(* Logix 5000 project; controller GEA_Test_Chamber vendor 1 type 14 code 196 rev 32.14; software revision 32.04; part 4 of 11 *)
(* tags used below, declared in another part *)
   Transaction : raC_UDT_ModbusClientTransaction;
   Wrk_Bit : DINT;
   Wrk_Byte : DINT;
(* raC_Tec_NetModbusTCPClient_BuildReqStr, continued *)

ROUTINE Prescan   (* ladder *)
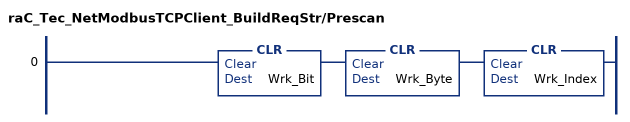
   0: CLR(Wrk_Bit)CLR(Wrk_Byte)CLR(Wrk_Index);
END_ROUTINE
END_ADD_ON_INSTRUCTION

ADD_ON_INSTRUCTION raC_Tec_NetModbusTCPClient_ChkWrReply   (* revision 2.0, ExecutePrescan *)
VAR_OUTPUT
   TransFound : BOOL; {access Read Only}
END_VAR
VAR_IN_OUT
   Transactions : raC_UDT_ModbusClientTransaction[5]; {required}
END_VAR
VAR_INPUT
   TransactionID : INT; {required}
   ModbusBytes : DINT; {required}
END_VAR
VAR_OUTPUT
   LocalOffset : INT; {access Read Only}
   Count : INT; {access Read Only}
END_VAR
VAR_INPUT
   Command : DINT; {required}
   LastTransaction : DINT; {required}
END_VAR
VAR
   Wrk_TransactionPtr : DINT; {access None}
END_VAR

ROUTINE Logic   (* ladder *)
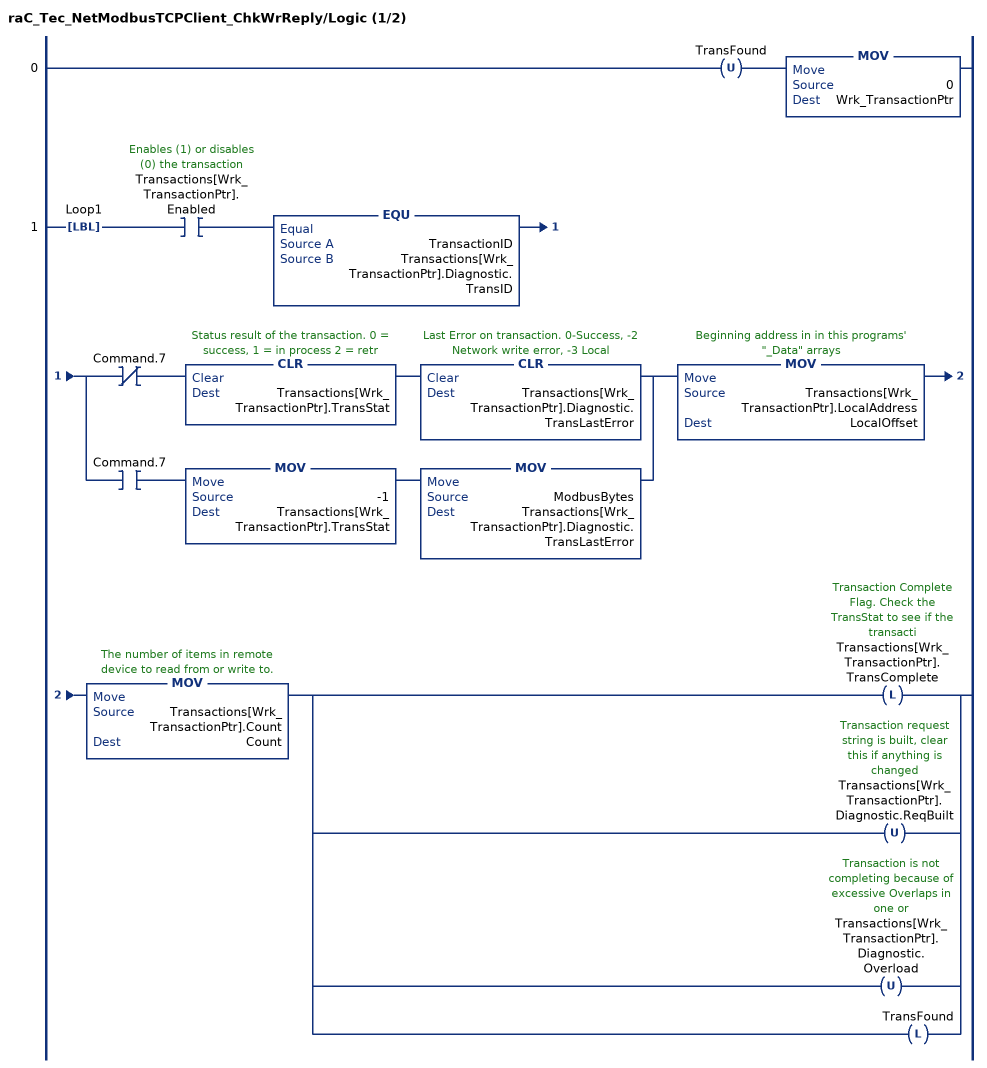
   0: OTU(TransFound)MOV(0,Wrk_TransactionPtr);
   1: LBL(Loop1)XIC(Transactions[Wrk_TransactionPtr].Enabled)EQU(TransactionID,Transactions[Wrk_TransactionPtr].Diagnostic.TransID)[XIO(Command.7) CLR(Transactions[Wrk_TransactionPtr].TransStat) CLR(Transactions[Wrk_TransactionPtr].Diagnostic.TransLastError) ,XIC(Command.7) MOV(-1,Transactions[Wrk_TransactionPtr].TransStat) MOV(ModbusBytes,Transactions[Wrk_TransactionPtr].Diagnostic.TransLastError) ]MOV(Transactions[Wrk_TransactionPtr].LocalAddress,LocalOffset)MOV(Transactions[Wrk_TransactionPtr].Count,Count)[OTL(Transactions[Wrk_TransactionPtr].TransComplete) ,OTU(Transactions[Wrk_TransactionPtr].Diagnostic.ReqBuilt) ,OTU(Transactions[Wrk_TransactionPtr].Diagnostic.Overload) ,OTL(TransFound) ];
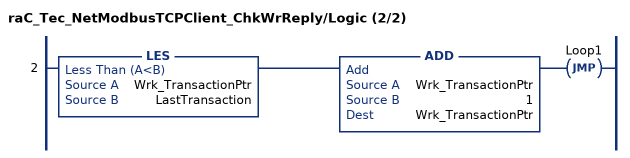
   2: LES(Wrk_TransactionPtr,LastTransaction)ADD(Wrk_TransactionPtr,1,Wrk_TransactionPtr)JMP(Loop1);
END_ROUTINE

ROUTINE Prescan   (* ladder *)
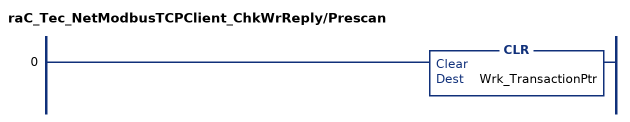
   0: CLR(Wrk_TransactionPtr);
END_ROUTINE
END_ADD_ON_INSTRUCTION

ADD_ON_INSTRUCTION raC_Tec_NetModbusTCPClient_RespStrBit   (* revision 2.0, ExecutePrescan *)
VAR_INPUT
   Inputs : BOOL; {required}
   Modbus_CMD_Len : INT; {required}
   LocalOffset : INT; {required}
END_VAR
VAR_IN_OUT
   ModbusData : raC_UDT_ModbusClientData; {required}
   CommandString : STR0462; {required}
END_VAR
VAR
   Wrk_BufferByteIndex : DINT; {access None}
   Wrk_Cmd_Last : INT; {access None}
   Wrk_Index : DINT; {access None}
   Wrk_BufferBitIndex : DINT; {access None}
   Wrk_ArraySize : DINT; {access None}
END_VAR

ROUTINE Logic   (* ladder *)
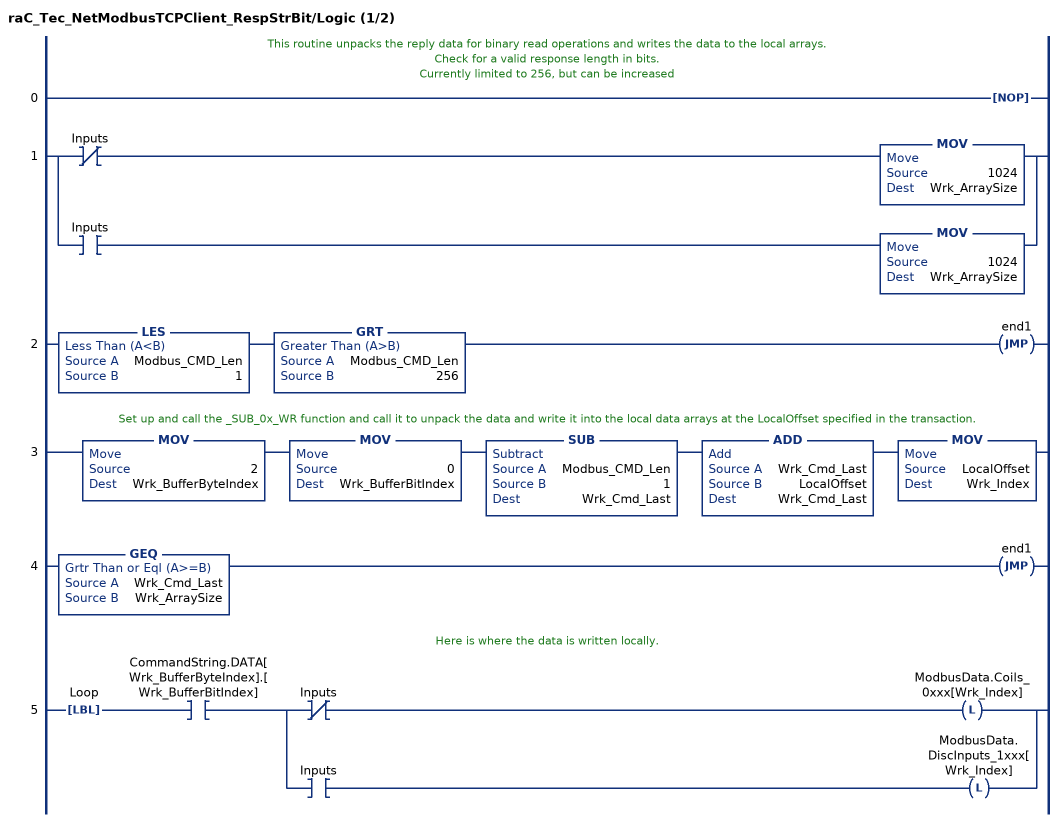
   // This routine unpacks the reply data for binary read operations and writes the data to the local arrays.
   // Check for a valid response length in bits.
   // Currently limited to 256, but can be increased
   0: NOP();
   1: [XIO(Inputs) MOV(1024,Wrk_ArraySize) ,XIC(Inputs) MOV(1024,Wrk_ArraySize) ];
   2: LES(Modbus_CMD_Len,1)GRT(Modbus_CMD_Len,256)JMP(end1);
   // Set up and call the _SUB_0x_WR function and call it to unpack the data and write it into the local data arrays at the LocalOffset specified in the transaction.
   3: MOV(2,Wrk_BufferByteIndex)MOV(0,Wrk_BufferBitIndex)SUB(Modbus_CMD_Len,1,Wrk_Cmd_Last)ADD(Wrk_Cmd_Last,LocalOffset,Wrk_Cmd_Last)MOV(LocalOffset,Wrk_Index);
   4: GEQ(Wrk_Cmd_Last,Wrk_ArraySize)JMP(end1);
   // Here is where the data is written locally.
   5: LBL(Loop)XIC(CommandString.DATA[Wrk_BufferByteIndex].[Wrk_BufferBitIndex])[XIO(Inputs) OTL(ModbusData.Coils_0xxx[Wrk_Index]) ,XIC(Inputs) OTL(ModbusData.DiscInputs_1xxx[Wrk_Index]) ];
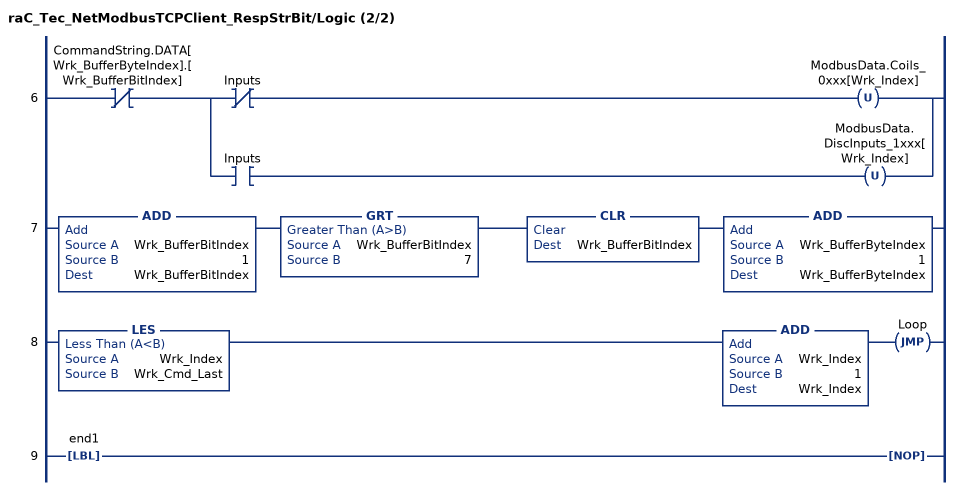
   6: XIO(CommandString.DATA[Wrk_BufferByteIndex].[Wrk_BufferBitIndex])[XIO(Inputs) OTU(ModbusData.Coils_0xxx[Wrk_Index]) ,XIC(Inputs) OTU(ModbusData.DiscInputs_1xxx[Wrk_Index]) ];
   7: ADD(Wrk_BufferBitIndex,1,Wrk_BufferBitIndex)GRT(Wrk_BufferBitIndex,7)CLR(Wrk_BufferBitIndex)ADD(Wrk_BufferByteIndex,1,Wrk_BufferByteIndex);
   8: LES(Wrk_Index,Wrk_Cmd_Last)ADD(Wrk_Index,1,Wrk_Index)JMP(Loop);
   9: LBL(end1)NOP();
END_ROUTINE

ROUTINE Prescan   (* ladder *)
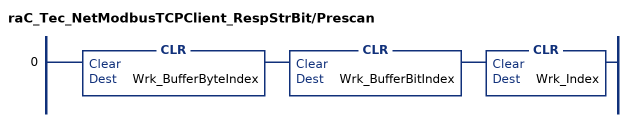
   0: CLR(Wrk_BufferByteIndex)CLR(Wrk_BufferBitIndex)CLR(Wrk_Index);
END_ROUTINE
END_ADD_ON_INSTRUCTION

ADD_ON_INSTRUCTION raC_Tec_NetModbusTCPClient_RespStrWord   (* revision 2.0, ExecutePrescan *)
VAR_INPUT
   Reg3xx : BOOL; {required}
   Modbus_CMD_Len : INT; {required}
   LocalOffset : INT; {required}
END_VAR
VAR_IN_OUT
   ModbusData : raC_UDT_ModbusClientData; {required}
   CommandString : STR0462; {required}
END_VAR
VAR
   Wrk_StringPosition : DINT; {access None}
   Wrk_Cmd_Last : INT; {access None}
   Wrk_Temp_Int : INT; {access None}
   Wrk_Index : DINT; {access None}
END_VAR

ROUTINE Logic   (* ladder *)
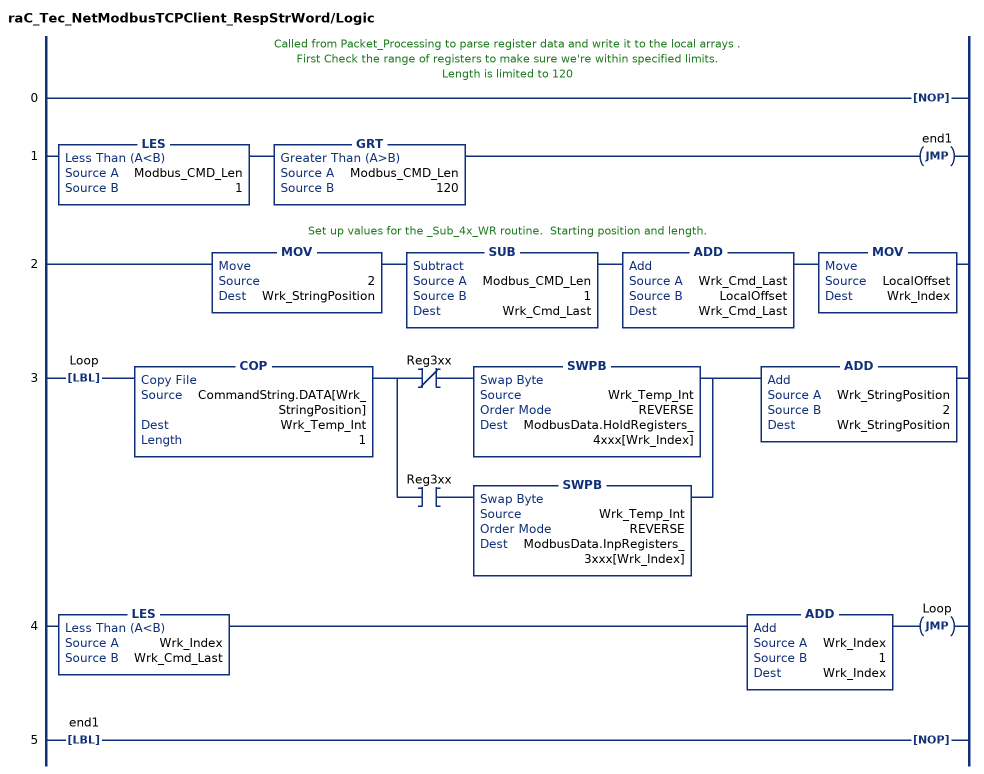
   // Called from Packet_Processing to parse register data and write it to the local arrays .
   // First Check the range of registers to make sure we're within specified limits.
   // Length is limited to 120
   0: NOP();
   1: LES(Modbus_CMD_Len,1)GRT(Modbus_CMD_Len,120)JMP(end1);
   // Set up values for the _Sub_4x_WR routine.  Starting position and length.
   2: MOV(2,Wrk_StringPosition)SUB(Modbus_CMD_Len,1,Wrk_Cmd_Last)ADD(Wrk_Cmd_Last,LocalOffset,Wrk_Cmd_Last)MOV(LocalOffset,Wrk_Index);
   3: LBL(Loop)COP(CommandString.DATA[Wrk_StringPosition],Wrk_Temp_Int,1)[XIO(Reg3xx) SWPB(Wrk_Temp_Int,REVERSE,ModbusData.HoldRegisters_4xxx[Wrk_Index]) ,XIC(Reg3xx) SWPB(Wrk_Temp_Int,REVERSE,ModbusData.InpRegisters_3xxx[Wrk_Index]) ]ADD(Wrk_StringPosition,2,Wrk_StringPosition);
   4: LES(Wrk_Index,Wrk_Cmd_Last)ADD(Wrk_Index,1,Wrk_Index)JMP(Loop);
   5: LBL(end1)NOP();
END_ROUTINE

ROUTINE Prescan   (* ladder *)
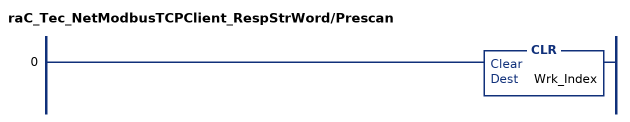
   0: CLR(Wrk_Index);
END_ROUTINE
END_ADD_ON_INSTRUCTION

ADD_ON_INSTRUCTION raC_Tec_NetModbusTCPServer_FndEmptySckt   (* revision 2.3 *)
VAR_INPUT
   NewInstance : DINT; {required}
   NewAddress : DINT; {required}
END_VAR
VAR_IN_OUT
   Sockets : raC_UDT_ModbusServerRWSocket[10]; {required}
END_VAR
VAR_OUTPUT
   Assigned : BOOL; {access Read Only, visible}
   NoRoom : BOOL; {access Read Only, visible}
END_VAR
VAR
   Wrk_InstIndex : DINT; {access None}
   Wrk_Size : DINT; {access None}
   Wrk_LastElement : DINT; {access None}
END_VAR

ROUTINE Logic   (* ladder *)
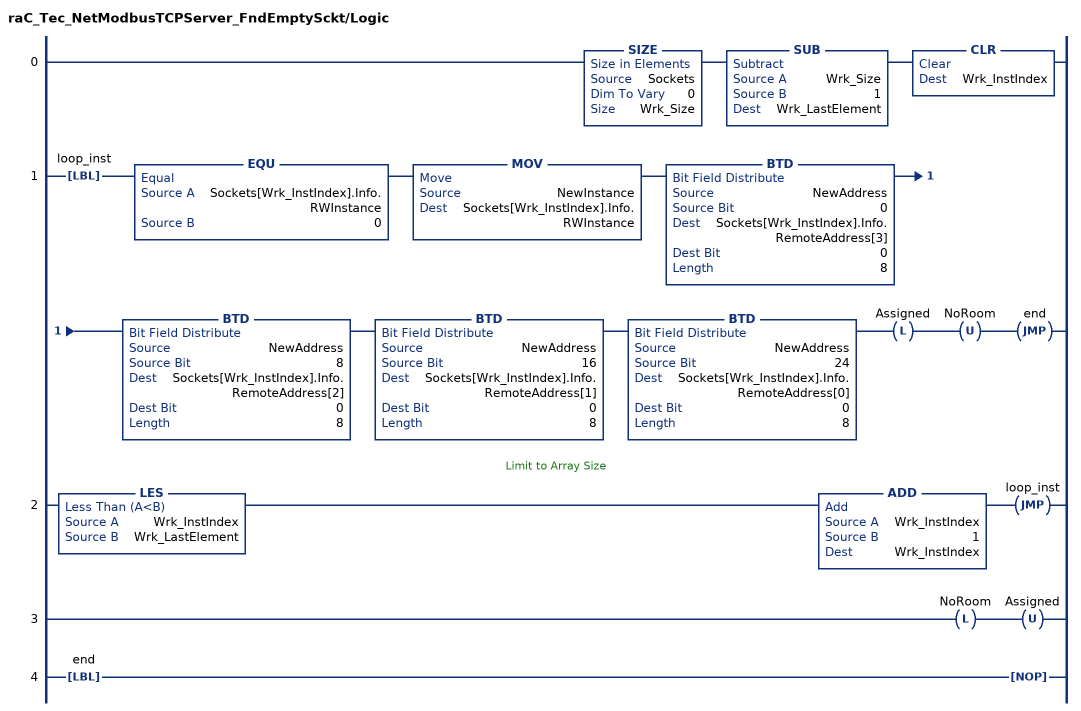
   0: SIZE(Sockets,0,Wrk_Size)SUB(Wrk_Size,1,Wrk_LastElement)CLR(Wrk_InstIndex);
   1: LBL(loop_inst)EQU(Sockets[Wrk_InstIndex].Info.RWInstance,0)MOV(NewInstance,Sockets[Wrk_InstIndex].Info.RWInstance)BTD(NewAddress,0,Sockets[Wrk_InstIndex].Info.RemoteAddress[3],0,8)BTD(NewAddress,8,Sockets[Wrk_InstIndex].Info.RemoteAddress[2],0,8)BTD(NewAddress,16,Sockets[Wrk_InstIndex].Info.RemoteAddress[1],0,8)BTD(NewAddress,24,Sockets[Wrk_InstIndex].Info.RemoteAddress[0],0,8)OTL(Assigned)OTU(NoRoom)JMP(end);
   // Limit to Array Size
   2: LES(Wrk_InstIndex,Wrk_LastElement)ADD(Wrk_InstIndex,1,Wrk_InstIndex)JMP(loop_inst);
   3: OTL(NoRoom)OTU(Assigned);
   4: LBL(end)NOP();
END_ROUTINE
END_ADD_ON_INSTRUCTION

ADD_ON_INSTRUCTION raC_Tec_NetModbusTCPServer_RespStrBit   (* revision 2.0, ExecutePrescan *)
VAR_INPUT
   Modbus_CMD_Start : INT; {required}
   Modbus_CMD_Len : INT; {required}
   Modbus_CMD : DINT; {required}
END_VAR
VAR_IN_OUT
   ModbusData : raC_UDT_ModbusServerData; {required}
   CommandString : STR0462; {required}
   ResponseString : STR0462; {required}
END_VAR
VAR
   Wrk_BufferByteIndex : DINT; {access None}
   Wrk_Cmd_Last : INT; {access None}
   Wrk_TempInt : INT; {access None}
   Wrk_Index : DINT; {access None}
   Wrk_BufferBitIndex : DINT; {access None}
   Wrk_Valid_Start : BOOL; {access None}
   Wrk_Valid_Len : BOOL; {access None}
   Wrk_Valid_Value_05 : BOOL; {access None}
   Wrk_Valid_End : BOOL; {access None}
   Wrk_CMD_END : DINT; {access None}
   Wrk_Valid_CMD1 : BOOL; {access None}
   Wrk_Valid_CMD2 : BOOL; {access None}
   Wrk_Valid_CMD15 : BOOL; {access None}
   Wrk_Valid_CMD5 : BOOL; {access None}
   Wrk_Byte_Count : DINT; {access None}
   Wrk_ret_CMD : STR0008; {access None}
   Wrk_ret_len : STR0008; {access None}
   Wrk_MbBitIndex : DINT; {access None}
   Wrk_TempInt1 : DINT; {access None}
   Wrk_AddrLimit : DINT; {access None}
   Wrk_MbBitIndex5 : DINT; {access None}
   Wrk_MbBitIndex15 : DINT; {access None}
END_VAR

ROUTINE Logic   (* ladder *)
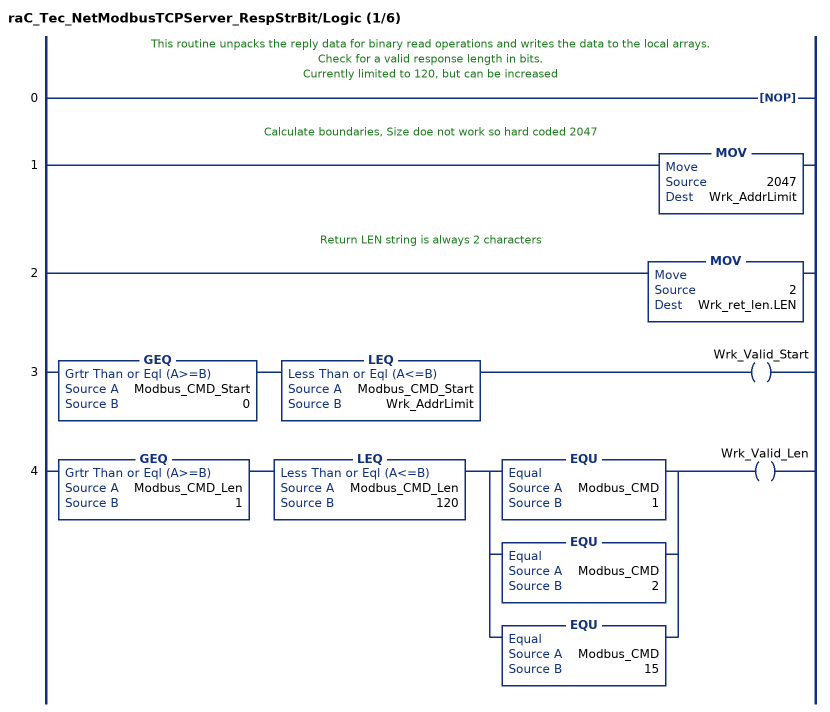
   // This routine unpacks the reply data for binary read operations and writes the data to the local arrays.
   // Check for a valid response length in bits.
   // Currently limited to 120, but can be increased
   0: NOP();
   // Calculate boundaries, Size doe not work so hard coded 2047
   1: MOV(2047,Wrk_AddrLimit);
   // Return LEN string is always 2 characters
   2: MOV(2,Wrk_ret_len.LEN);
   3: GEQ(Modbus_CMD_Start,0)LEQ(Modbus_CMD_Start,Wrk_AddrLimit)OTE(Wrk_Valid_Start);
   4: GEQ(Modbus_CMD_Len,1)LEQ(Modbus_CMD_Len,120)[EQU(Modbus_CMD,1) ,EQU(Modbus_CMD,2) ,EQU(Modbus_CMD,15) ]OTE(Wrk_Valid_Len);
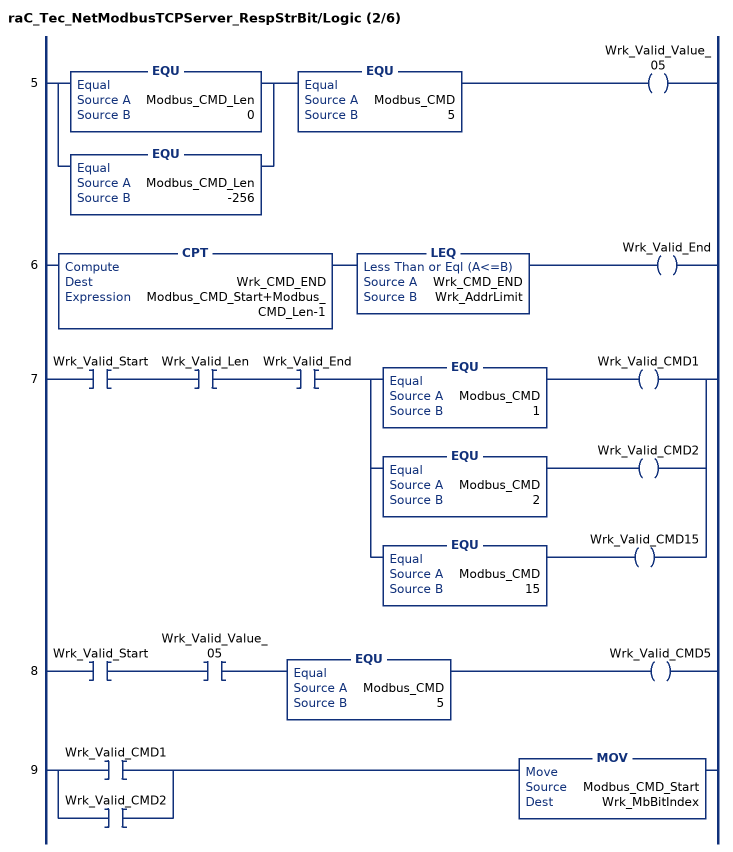
   5: [EQU(Modbus_CMD_Len,0) ,EQU(Modbus_CMD_Len,-256) ]EQU(Modbus_CMD,5)OTE(Wrk_Valid_Value_05);
   6: CPT(Wrk_CMD_END,Modbus_CMD_Start+Modbus_CMD_Len-1)LEQ(Wrk_CMD_END,Wrk_AddrLimit)OTE(Wrk_Valid_End);
   7: XIC(Wrk_Valid_Start)XIC(Wrk_Valid_Len)XIC(Wrk_Valid_End)[EQU(Modbus_CMD,1) OTE(Wrk_Valid_CMD1) ,EQU(Modbus_CMD,2) OTE(Wrk_Valid_CMD2) ,EQU(Modbus_CMD,15) OTE(Wrk_Valid_CMD15) ];
   8: XIC(Wrk_Valid_Start)XIC(Wrk_Valid_Value_05)EQU(Modbus_CMD,5)OTE(Wrk_Valid_CMD5);
   9: [XIC(Wrk_Valid_CMD1) ,XIC(Wrk_Valid_CMD2) ]MOV(Modbus_CMD_Start,Wrk_MbBitIndex);
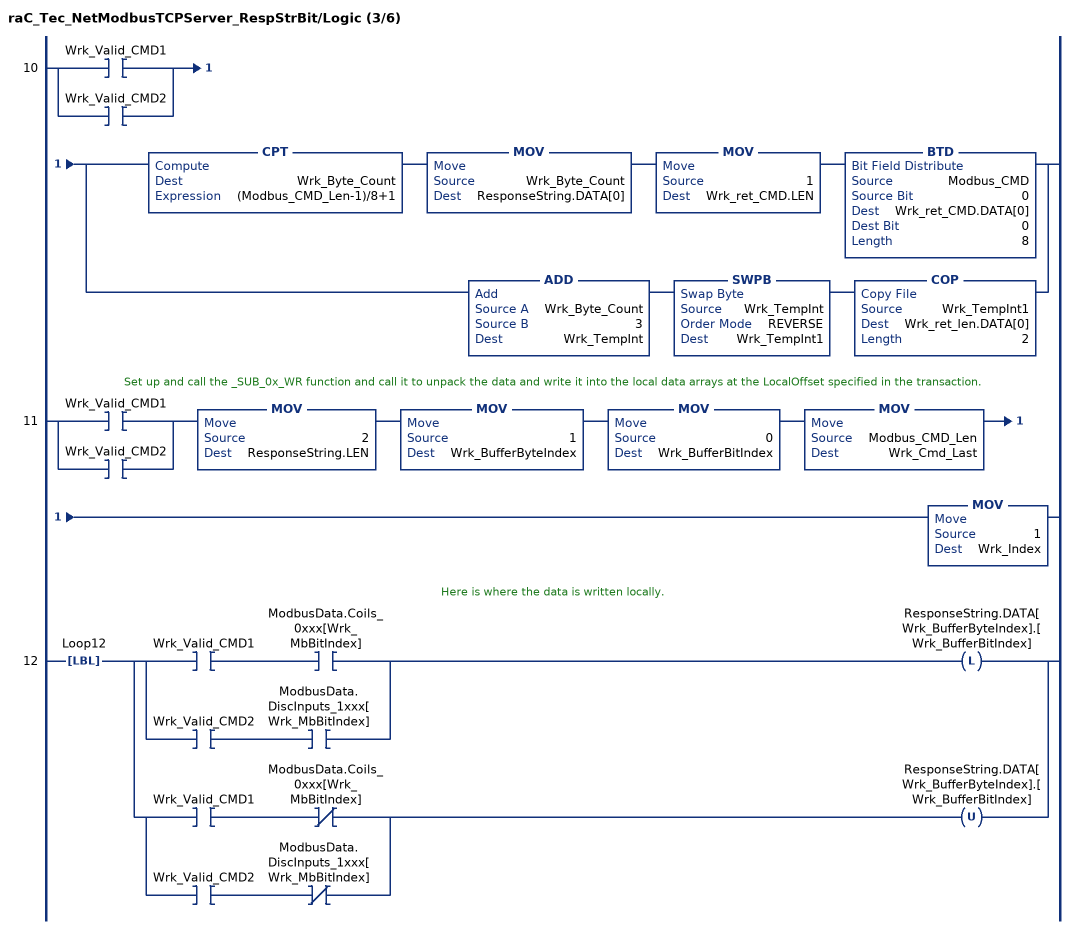
   10: [XIC(Wrk_Valid_CMD1) ,XIC(Wrk_Valid_CMD2) ][CPT(Wrk_Byte_Count,(Modbus_CMD_Len-1)/8+1) MOV(Wrk_Byte_Count,ResponseString.DATA[0]) MOV(1,Wrk_ret_CMD.LEN) BTD(Modbus_CMD,0,Wrk_ret_CMD.DATA[0],0,8) ,ADD(Wrk_Byte_Count,3,Wrk_TempInt) SWPB(Wrk_TempInt,REVERSE,Wrk_TempInt1) COP(Wrk_TempInt1,Wrk_ret_len.DATA[0],2) ];
   // Set up and call the _SUB_0x_WR function and call it to unpack the data and write it into the local data arrays at the LocalOffset specified in the transaction.
   11: [XIC(Wrk_Valid_CMD1) ,XIC(Wrk_Valid_CMD2) ]MOV(2,ResponseString.LEN)MOV(1,Wrk_BufferByteIndex)MOV(0,Wrk_BufferBitIndex)MOV(Modbus_CMD_Len,Wrk_Cmd_Last)MOV(1,Wrk_Index);
   // Here is where the data is written locally.
   12: LBL(Loop12)[[XIC(Wrk_Valid_CMD1) XIC(ModbusData.Coils_0xxx[Wrk_MbBitIndex]) ,XIC(Wrk_Valid_CMD2) XIC(ModbusData.DiscInputs_1xxx[Wrk_MbBitIndex]) ] OTL(ResponseString.DATA[Wrk_BufferByteIndex].[Wrk_BufferBitIndex]) ,[XIC(Wrk_Valid_CMD1) XIO(ModbusData.Coils_0xxx[Wrk_MbBitIndex]) ,XIC(Wrk_Valid_CMD2) XIO(ModbusData.DiscInputs_1xxx[Wrk_MbBitIndex]) ] OTU(ResponseString.DATA[Wrk_BufferByteIndex].[Wrk_BufferBitIndex]) ];
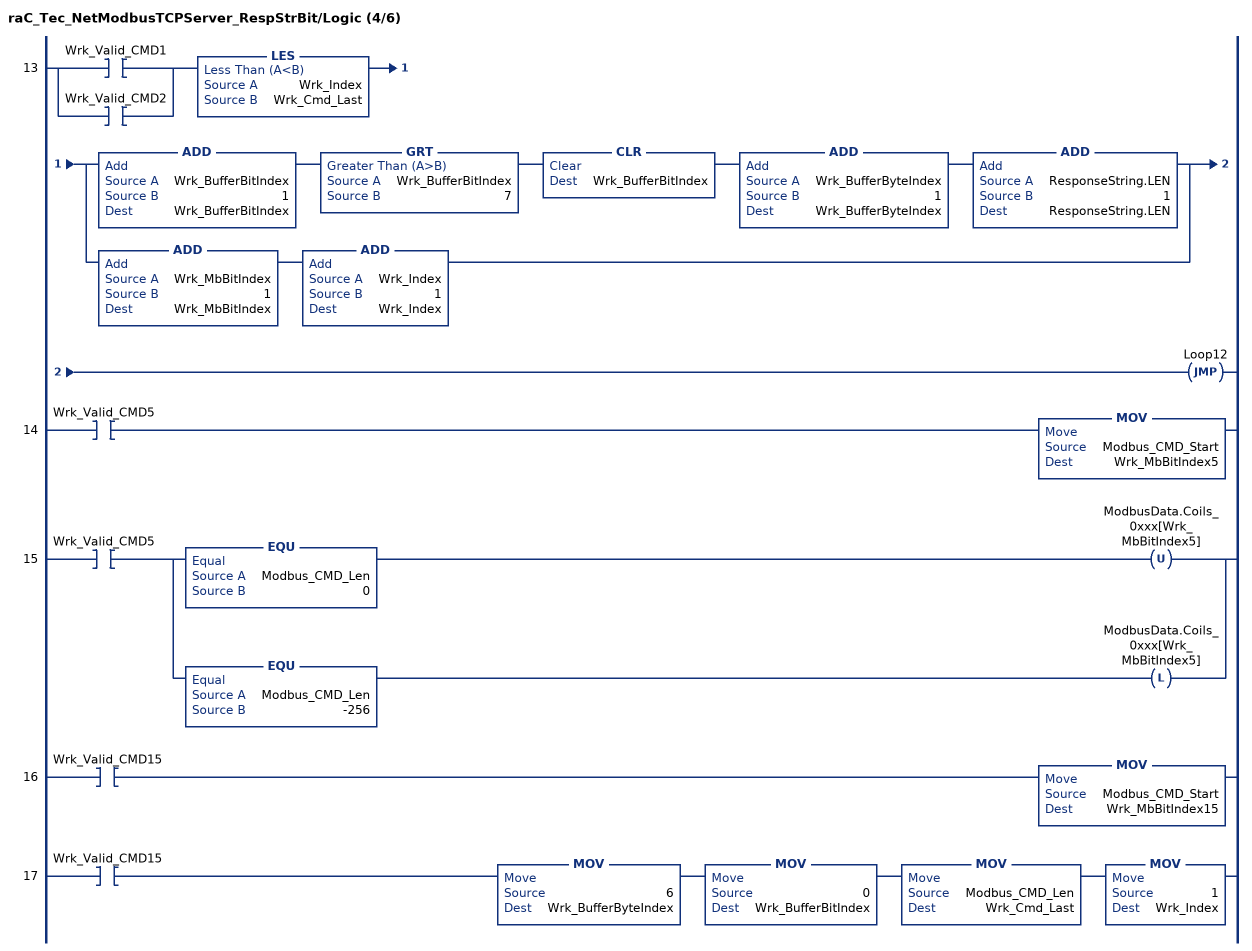
   13: [XIC(Wrk_Valid_CMD1) ,XIC(Wrk_Valid_CMD2) ]LES(Wrk_Index,Wrk_Cmd_Last)[ADD(Wrk_BufferBitIndex,1,Wrk_BufferBitIndex) GRT(Wrk_BufferBitIndex,7) CLR(Wrk_BufferBitIndex) ADD(Wrk_BufferByteIndex,1,Wrk_BufferByteIndex) ADD(ResponseString.LEN,1,ResponseString.LEN) ,ADD(Wrk_MbBitIndex,1,Wrk_MbBitIndex) ADD(Wrk_Index,1,Wrk_Index) ]JMP(Loop12);
   14: XIC(Wrk_Valid_CMD5)MOV(Modbus_CMD_Start,Wrk_MbBitIndex5);
   15: XIC(Wrk_Valid_CMD5)[EQU(Modbus_CMD_Len,0) OTU(ModbusData.Coils_0xxx[Wrk_MbBitIndex5]) ,EQU(Modbus_CMD_Len,-256) OTL(ModbusData.Coils_0xxx[Wrk_MbBitIndex5]) ];
   16: XIC(Wrk_Valid_CMD15)MOV(Modbus_CMD_Start,Wrk_MbBitIndex15);
   17: XIC(Wrk_Valid_CMD15)MOV(6,Wrk_BufferByteIndex)MOV(0,Wrk_BufferBitIndex)MOV(Modbus_CMD_Len,Wrk_Cmd_Last)MOV(1,Wrk_Index);
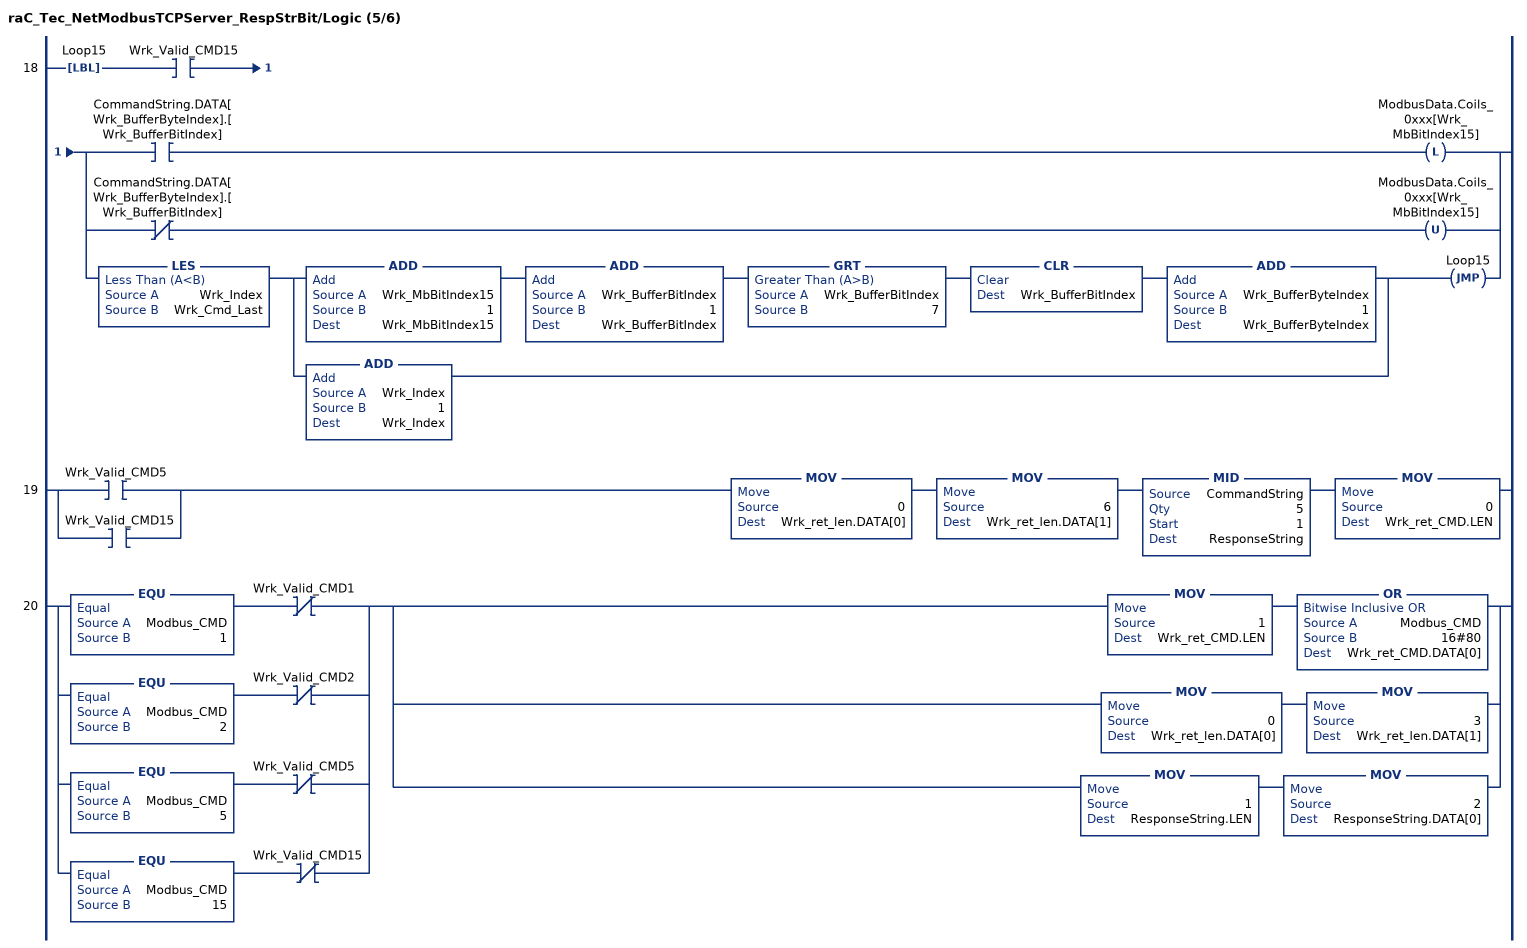
   18: LBL(Loop15)XIC(Wrk_Valid_CMD15)[[XIC(CommandString.DATA[Wrk_BufferByteIndex].[Wrk_BufferBitIndex]) OTL(ModbusData.Coils_0xxx[Wrk_MbBitIndex15]) ,XIO(CommandString.DATA[Wrk_BufferByteIndex].[Wrk_BufferBitIndex]) OTU(ModbusData.Coils_0xxx[Wrk_MbBitIndex15]) ] ,LES(Wrk_Index,Wrk_Cmd_Last) [ADD(Wrk_MbBitIndex15,1,Wrk_MbBitIndex15) ADD(Wrk_BufferBitIndex,1,Wrk_BufferBitIndex) GRT(Wrk_BufferBitIndex,7) CLR(Wrk_BufferBitIndex) ADD(Wrk_BufferByteIndex,1,Wrk_BufferByteIndex) ,ADD(Wrk_Index,1,Wrk_Index) ] JMP(Loop15) ];
   19: [XIC(Wrk_Valid_CMD5) ,XIC(Wrk_Valid_CMD15) ]MOV(0,Wrk_ret_len.DATA[0])MOV(6,Wrk_ret_len.DATA[1])MID(CommandString,5,1,ResponseString)MOV(0,Wrk_ret_CMD.LEN);
   20: [EQU(Modbus_CMD,1) XIO(Wrk_Valid_CMD1) ,EQU(Modbus_CMD,2) XIO(Wrk_Valid_CMD2) ,EQU(Modbus_CMD,5) XIO(Wrk_Valid_CMD5) ,EQU(Modbus_CMD,15) XIO(Wrk_Valid_CMD15) ][MOV(1,Wrk_ret_CMD.LEN) OR(Modbus_CMD,16#80,Wrk_ret_CMD.DATA[0]) ,MOV(0,Wrk_ret_len.DATA[0]) MOV(3,Wrk_ret_len.DATA[1]) ,MOV(1,ResponseString.LEN) MOV(2,ResponseString.DATA[0]) ];
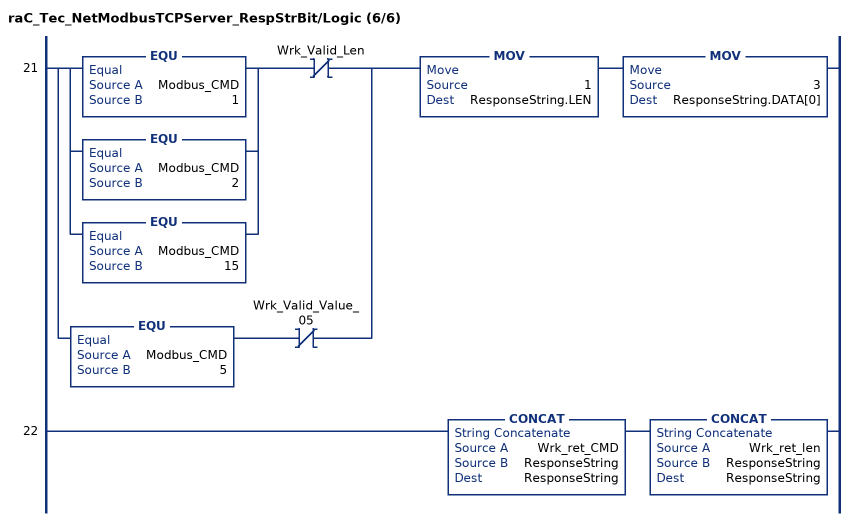
   21: [[EQU(Modbus_CMD,1) ,EQU(Modbus_CMD,2) ,EQU(Modbus_CMD,15) ] XIO(Wrk_Valid_Len) ,EQU(Modbus_CMD,5) XIO(Wrk_Valid_Value_05) ]MOV(1,ResponseString.LEN)MOV(3,ResponseString.DATA[0]);
   22: CONCAT(Wrk_ret_CMD,ResponseString,ResponseString)CONCAT(Wrk_ret_len,ResponseString,ResponseString);
END_ROUTINE

ROUTINE Prescan   (* ladder *)
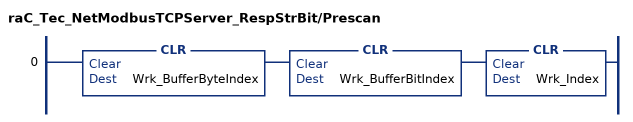
   0: CLR(Wrk_BufferByteIndex)CLR(Wrk_BufferBitIndex)CLR(Wrk_Index);
END_ROUTINE
END_ADD_ON_INSTRUCTION

ADD_ON_INSTRUCTION raC_Tec_NetModbusTCPServer_RespStrWord   (* revision 2.0, ExecutePrescan *)
VAR_INPUT
   Modbus_CMD_Start : INT; {required}
   Modbus_CMD_Len : INT; {required}
   Modbus_CMD : DINT; {required}
END_VAR
VAR_IN_OUT
   ModbusData : raC_UDT_ModbusServerData; {required}
   CommandString : STR0462; {required}
   ResponseString : STR0462; {required}
END_VAR
VAR
   Wrk_Cmd_Last : INT; {access None}
   Wrk_ByteCount : INT; {access None}
   Wrk_Index : DINT; {access None}
   Wrk_Valid_Start : BOOL; {access None}
   Wrk_Valid_Len : BOOL; {access None}
   Wrk_ret_len : STR0008; {access None}
   Wrk_TempInt : INT; {access None}
   Wrk_Valid_Len_16 : BOOL; {access None}
   Wrk_CMD_End : DINT; {access None}
   Wrk_Valid_end : BOOL; {access None}
   Wrk_Valid_CMD3 : BOOL; {access None}
   Wrk_Valid_CMD4 : BOOL; {access None}
   Wrk_Valid_CMD16 : BOOL; {access None}
   Wrk_Valid_CMD6 : BOOL; {access None}
   Wrk_ret_CMD : STR0008; {access None}
   Wrk_StrPos : DINT; {access None}
   Wrk_Size4x : DINT; {access None}
   Wrk_Size3x : DINT; {access None}
   Wrk_AddrLimit : DINT; {access None}
   Wrk_TempByteLength : DINT; {access None}
END_VAR

ROUTINE Logic   (* ladder *)
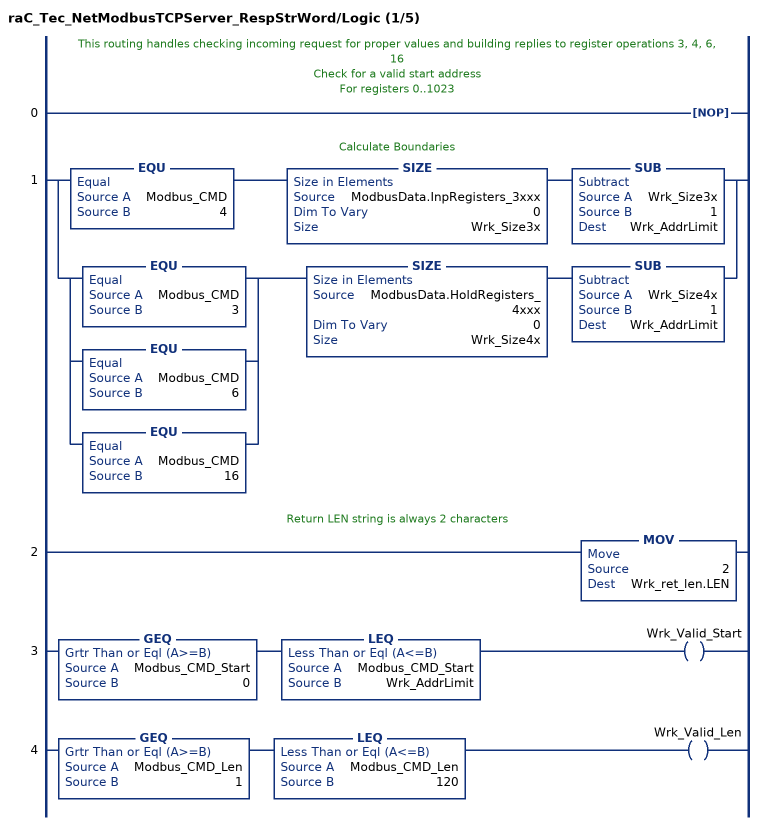
   // This routing handles checking incoming request for proper values and building replies to register operations 3, 4, 6, 16
   // Check for a valid start address
   // For registers 0..1023
   0: NOP();
   // Calculate Boundaries
   1: [EQU(Modbus_CMD,4) SIZE(ModbusData.InpRegisters_3xxx,0,Wrk_Size3x) SUB(Wrk_Size3x,1,Wrk_AddrLimit) ,[EQU(Modbus_CMD,3) ,EQU(Modbus_CMD,6) ,EQU(Modbus_CMD,16) ] SIZE(ModbusData.HoldRegisters_4xxx,0,Wrk_Size4x) SUB(Wrk_Size4x,1,Wrk_AddrLimit) ];
   // Return LEN string is always 2 characters
   2: MOV(2,Wrk_ret_len.LEN);
   3: GEQ(Modbus_CMD_Start,0)LEQ(Modbus_CMD_Start,Wrk_AddrLimit)OTE(Wrk_Valid_Start);
   4: GEQ(Modbus_CMD_Len,1)LEQ(Modbus_CMD_Len,120)OTE(Wrk_Valid_Len);
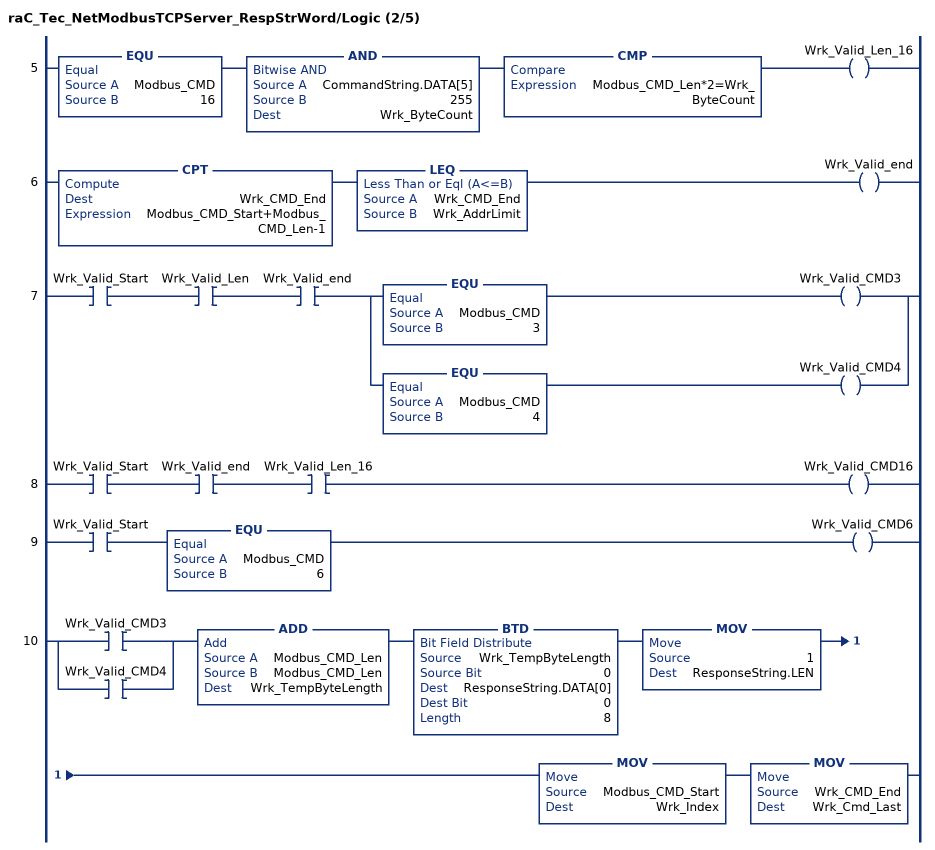
   5: EQU(Modbus_CMD,16)AND(CommandString.DATA[5],255,Wrk_ByteCount)CMP(Modbus_CMD_Len*2=Wrk_ByteCount)OTE(Wrk_Valid_Len_16);
   6: CPT(Wrk_CMD_End,Modbus_CMD_Start+Modbus_CMD_Len-1)LEQ(Wrk_CMD_End,Wrk_AddrLimit)OTE(Wrk_Valid_end);
   7: XIC(Wrk_Valid_Start)XIC(Wrk_Valid_Len)XIC(Wrk_Valid_end)[EQU(Modbus_CMD,3) OTE(Wrk_Valid_CMD3) ,EQU(Modbus_CMD,4) OTE(Wrk_Valid_CMD4) ];
   8: XIC(Wrk_Valid_Start)XIC(Wrk_Valid_end)XIC(Wrk_Valid_Len_16)OTE(Wrk_Valid_CMD16);
   9: XIC(Wrk_Valid_Start)EQU(Modbus_CMD,6)OTE(Wrk_Valid_CMD6);
   10: [XIC(Wrk_Valid_CMD3) ,XIC(Wrk_Valid_CMD4) ]ADD(Modbus_CMD_Len,Modbus_CMD_Len,Wrk_TempByteLength)BTD(Wrk_TempByteLength,0,ResponseString.DATA[0],0,8)MOV(1,ResponseString.LEN)MOV(Modbus_CMD_Start,Wrk_Index)MOV(Wrk_CMD_End,Wrk_Cmd_Last);
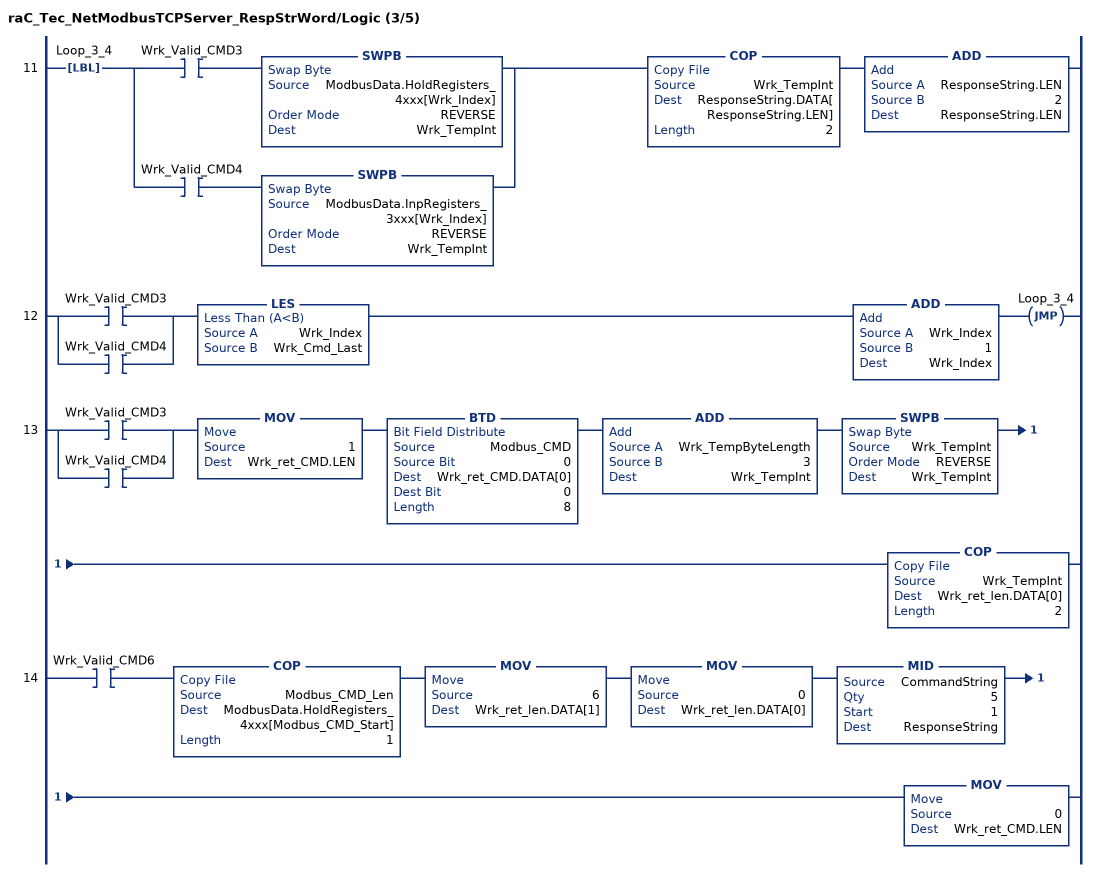
   11: LBL(Loop_3_4)[XIC(Wrk_Valid_CMD3) SWPB(ModbusData.HoldRegisters_4xxx[Wrk_Index],REVERSE,Wrk_TempInt) ,XIC(Wrk_Valid_CMD4) SWPB(ModbusData.InpRegisters_3xxx[Wrk_Index],REVERSE,Wrk_TempInt) ]COP(Wrk_TempInt,ResponseString.DATA[ResponseString.LEN],2)ADD(ResponseString.LEN,2,ResponseString.LEN);
   12: [XIC(Wrk_Valid_CMD3) ,XIC(Wrk_Valid_CMD4) ]LES(Wrk_Index,Wrk_Cmd_Last)ADD(Wrk_Index,1,Wrk_Index)JMP(Loop_3_4);
   13: [XIC(Wrk_Valid_CMD3) ,XIC(Wrk_Valid_CMD4) ]MOV(1,Wrk_ret_CMD.LEN)BTD(Modbus_CMD,0,Wrk_ret_CMD.DATA[0],0,8)ADD(Wrk_TempByteLength,3,Wrk_TempInt)SWPB(Wrk_TempInt,REVERSE,Wrk_TempInt)COP(Wrk_TempInt,Wrk_ret_len.DATA[0],2);
   14: XIC(Wrk_Valid_CMD6)COP(Modbus_CMD_Len,ModbusData.HoldRegisters_4xxx[Modbus_CMD_Start],1)MOV(6,Wrk_ret_len.DATA[1])MOV(0,Wrk_ret_len.DATA[0])MID(CommandString,5,1,ResponseString)MOV(0,Wrk_ret_CMD.LEN);
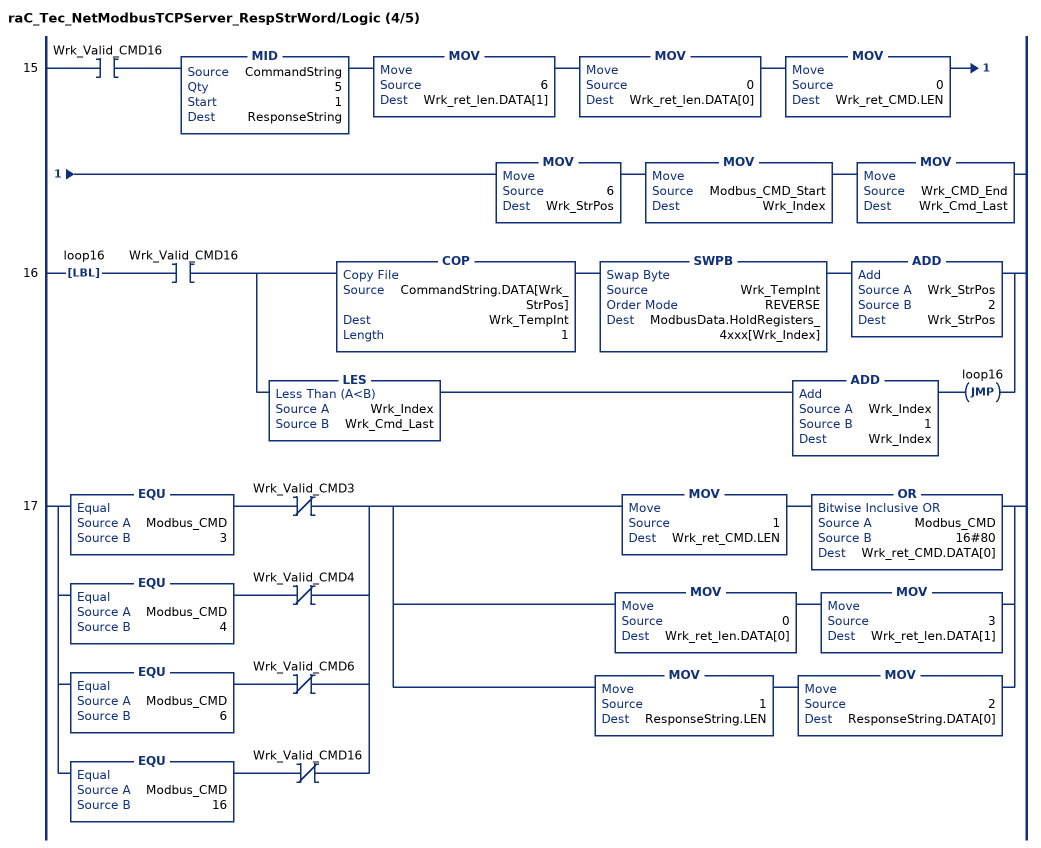
   15: XIC(Wrk_Valid_CMD16)MID(CommandString,5,1,ResponseString)MOV(6,Wrk_ret_len.DATA[1])MOV(0,Wrk_ret_len.DATA[0])MOV(0,Wrk_ret_CMD.LEN)MOV(6,Wrk_StrPos)MOV(Modbus_CMD_Start,Wrk_Index)MOV(Wrk_CMD_End,Wrk_Cmd_Last);
   16: LBL(loop16)XIC(Wrk_Valid_CMD16)[COP(CommandString.DATA[Wrk_StrPos],Wrk_TempInt,1) SWPB(Wrk_TempInt,REVERSE,ModbusData.HoldRegisters_4xxx[Wrk_Index]) ADD(Wrk_StrPos,2,Wrk_StrPos) ,LES(Wrk_Index,Wrk_Cmd_Last) ADD(Wrk_Index,1,Wrk_Index) JMP(loop16) ];
   17: [EQU(Modbus_CMD,3) XIO(Wrk_Valid_CMD3) ,EQU(Modbus_CMD,4) XIO(Wrk_Valid_CMD4) ,EQU(Modbus_CMD,6) XIO(Wrk_Valid_CMD6) ,EQU(Modbus_CMD,16) XIO(Wrk_Valid_CMD16) ][MOV(1,Wrk_ret_CMD.LEN) OR(Modbus_CMD,16#80,Wrk_ret_CMD.DATA[0]) ,MOV(0,Wrk_ret_len.DATA[0]) MOV(3,Wrk_ret_len.DATA[1]) ,MOV(1,ResponseString.LEN) MOV(2,ResponseString.DATA[0]) ];
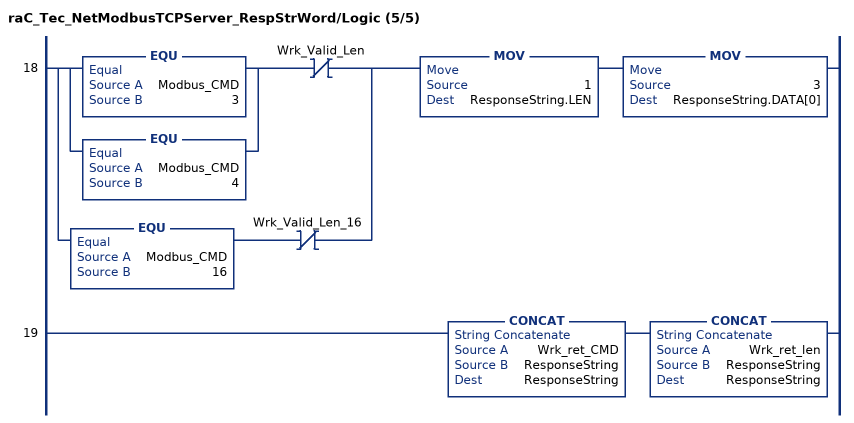
   18: [[EQU(Modbus_CMD,3) ,EQU(Modbus_CMD,4) ] XIO(Wrk_Valid_Len) ,EQU(Modbus_CMD,16) XIO(Wrk_Valid_Len_16) ]MOV(1,ResponseString.LEN)MOV(3,ResponseString.DATA[0]);
   19: CONCAT(Wrk_ret_CMD,ResponseString,ResponseString)CONCAT(Wrk_ret_len,ResponseString,ResponseString);
END_ROUTINE
